PROGRAM PRG_TEST
VAR
END_VAR

END_PROGRAM

(* stored: Version 1.1.0.1, ProductVersion 3.1.4024.9
   POU PRG_TEST: Id {55b693b2-7ec3-4123-bf43-681ce4807bf9}, SpecialFunc None *)
